Staubli VAL3: onEdit.pgx

public program onEdit(string& x_sItem[])
  local num l_nX
  local num l_nY
  local num l_nDelay
  local bool l_bValide
begin
  // convert to a num
  l_bValide=true
  toNum(x_sItem,l_nDelay,l_bValide)
  // change the field
  call use:insertDialog("DELAY [Sec] ",l_nDelay,0,100)
  // give back
  if l_nDelay>0
    if round(l_nDelay)==l_nDelay
      x_sItem=toString("",l_nDelay)
    else
      x_sItem=toString(".2",l_nDelay)
    endIf
  endIf
end
